FUNCTION_BLOCK FB_MoveAbsoluteNC_TestDouble IMPLEMENTS I_MoveAbsolute
VAR_INPUT
END_VAR
VAR_OUTPUT
END_VAR
VAR
END_VAR

{warning 'Add property implementation'}
PROPERTY Aborted : BOOL
GET
END_GET
END_PROPERTY

{warning 'Add property implementation'}
PROPERTY Active : BOOL
GET
END_GET
END_PROPERTY

{warning 'Add property implementation'}
PROPERTY Busy : BOOL
GET
END_GET
END_PROPERTY

{warning 'Add property implementation'}
PROPERTY CommandMoveAbsolute : BOOL
SET
END_SET
END_PROPERTY

{warning 'Add property implementation'}
PROPERTY Done : BOOL
GET
END_GET
END_PROPERTY

{warning 'Add property implementation'}
PROPERTY Error : BOOL
GET
END_GET
END_PROPERTY

{warning 'Add property implementation'}
PROPERTY ErrorID : UDINT
GET
END_GET
END_PROPERTY

{warning 'Add property implementation'}
PROPERTY Message : T_MAXSTRING
GET
END_GET
END_PROPERTY

{warning 'Add method implementation '}
METHOD MoveAbsolute
VAR_INPUT
    Position	: LREAL;
    Velocity	: LREAL;
    Acceleration	: LREAL := 0;
    Deceleration	: LREAL := 0;
    Jerk	: LREAL := 0;
    BufferMode	: MC_BufferMode := .MC_BufferMode.MC_Aborting;
END_VAR
END_METHOD

END_FUNCTION_BLOCK

(* stored: Version 1.1.0.1
   POU FB_MoveAbsoluteNC_TestDouble: Id {a1299b88-c1cc-47e6-86d2-69eec76abb7c}, SpecialFunc None
   Property Aborted: Id {d4e3cd51-5fee-4db6-8208-a2bc7e9fdd7a}
   Get Get: Id {26c0c97b-2d18-473c-9b75-fe721f82f49f}
   Property Active: Id {09738852-52fb-4077-a45f-6ebfef7b4a86}
   Get Get: Id {5e775f9a-a8f6-4a42-974f-288cf114ff26}
   Property Busy: Id {39175115-a127-49c4-80ac-dffa8f64dda2}
   Get Get: Id {5ac749c2-ac2c-41cb-a308-ca6e922fd588}
   Property CommandMoveAbsolute: Id {9eb83c04-aa48-4f9f-a6a7-3768920423d4}
   Set Set: Id {d7d59388-2f0d-423e-82ff-f43ef092b308}
   Property Done: Id {6c26a443-e660-4fcf-999f-11731e43cb8f}
   Get Get: Id {e1981ecc-2030-40ce-9a7c-d8a1d2e391e3}
   Property Error: Id {bd80d191-eec2-449f-96a3-3506f67108a1}
   Get Get: Id {0ea3b5eb-6486-46c5-902c-adf45a253412}
   Property ErrorID: Id {c366e1bd-70a4-48f4-838b-8982d7690ce1}
   Get Get: Id {0ef34ba1-602b-4eac-8648-615a36e3bda6}
   Property Message: Id {682bc89a-ba45-4a9c-bd43-aa24d1d42359}
   Get Get: Id {ad285937-0e0d-43a8-965c-8779c9795f7b}
   Method MoveAbsolute: Id {9d7d7069-91ef-47be-85d8-0bfdfbbff977} *)
